FUNCTION_BLOCK C_RESTFUL_SERVER
VAR_INPUT
END_VAR
VAR_OUTPUT
END_VAR
VAR
END_VAR

END_FUNCTION_BLOCK

(* stored: Version 1.1.0.1, ProductVersion 3.1.4019.2
   POU C_RESTFUL_SERVER: Id {2ed9c24a-91ed-4ae7-bf9b-56c52a3bf700}, SpecialFunc None *)
